// WARNING CODE //
	FB_AlarmCodeManager(
		bAlarm1			:= FALSE,   							//
		bAlarm2			:= FALSE, 								// 
		bAlarm3			:= FALSE, 								// 
		bAlarm4			:= FALSE, 								// 
		bAlarm5			:= FALSE,    							// 
		bAlarm6			:= FALSE, 								// 
		bAlarm7			:= FALSE, 								// 
		bAlarm8			:= FALSE, 								// 
		bAlarm9			:= FALSE,    							// 
		bAlarm10		:= FALSE, 								// 
		bAlarm11		:= FALSE, 								// 
		bAlarm12		:= FALSE, 								// 
		bAlarm13		:= FALSE,     							//
		bAlarm14		:= FALSE,  								//
		bAlarm15		:= FALSE,  								//
		wAlarmCode		=>MesDataExd.MesData.MesWarningCode);

// EVENT CODE //
	FB_AlarmCodeManager(
		bAlarm1			:= TON_Fermeture.Q AND NOT PT_Unlock_Alarm.Q, 	// Intrusion Detected
		bAlarm2			:= FALSE, 										// 
		bAlarm3			:= FALSE, 										// 
		bAlarm4			:= FALSE, 										// 
		bAlarm5			:= FALSE,    									// 
		bAlarm6			:= FALSE, 										// 
		bAlarm7			:= FALSE, 										// 
		bAlarm8			:= FALSE, 										// 
		bAlarm9			:= FALSE,    									// 
		bAlarm10		:= FALSE, 										// 
		bAlarm11		:= FALSE, 										// 
		bAlarm12		:= FALSE, 										// 
		bAlarm13		:= FALSE,     									// 
		bAlarm14		:= FALSE,  										// 
		bAlarm15		:= FALSE,  										// 
		wAlarmCode		=>MesDataExd.MesData.MesEventCode);
		
// When the alarm is activated for the first time, it is disabled for the duration of ParamTempoUnlockAlarm to avoid spamming alarms

PT_Unlock_Alarm(IN := TON_Fermeture.Q, PT := ParamTempoUnlockAlarm);
END_METHOD

METHOD M_Execute
//////////////////
//  Method Calls 
/////////////////

VAR 
	// Method local variables (reinitialized at each cycle) 
	
END_VAR

SUPER^.M_Execute() ;
END_METHOD

METHOD M_StateManager
//////////////////
// Detect when fire occurs
/////////////////

VAR 
	// Method local variables (reinitialized at each cycle)
 	MesStateInterm1 : BOOL;
	MesStateInterm2 : BOOL;
END_VAR

IF ParamCableCutSecurity THEN
	MesStateInterm1 := NOT IN_MesState1_IO ; 
	MesStateInterm2 := NOT IN_MesState2_IO ; 
ELSE 
	MesStateInterm1 := IN_MesState1_IO;
	MesStateInterm2 := IN_MesState2_IO;
END_IF

IF ParamNbSensors = 1 THEN 
	MesStateInterm2 := MesStateInterm1 ;
END_IF

IF ParamAtleastOne THEN 
MesDataExd.MesData.MesAlarmState := MesStateInterm1 OR MesStateInterm2 ; 
ELSE
MesDataExd.MesData.MesAlarmState := MesStateInterm1 AND MesStateInterm2 ; 
END_IF

R_TRIGAlarm(CLK:= MesDataExd.MesData.MesAlarmState ) ; 
IF R_TRIGAlarm.Q THEN
	MesCountAlarm :=  MIN(MesCountAlarm + 1 ,4294967295 ) ; 
ELSIF IN_ResetCounter THEN 
	MesCountAlarm := 0 ; 
END_IF

MesDataExd.MesData.MesCountAlarm	:= MesCountAlarm ;
END_METHOD

END_FUNCTION_BLOCK

// ---- 01_Equipement_Library/Sensors/TOR/FB_TOR_Spd.TcPOU
FUNCTION_BLOCK FB_TOR_Spd EXTENDS FB_TOR_Base
//////////////////
//  Surge Protection Device
//////////////////
VAR_INPUT PERSISTENT
	// Parameters of the Object (instance/model specific) 
	ParamTempoEs :TIME:=T#5S;(*  (s)Tempo before raising an alarm*)
END_VAR

VAR_OUTPUT
	//Child objects
	
END_VAR

VAR_INPUT
	// I/O Inputs 		                                     				
		
	
END_VAR

VAR
	//M_ALARMMANAGEMENT VARIABLES//
		FB_PermAlarm				: SR ;					// (NA) FB to maintain Fire Alarm even if sensor stop detection (burn) .
		TON_ES						: TON ; 
 
	//M_STATEMANAGER VARIABLES//
		MesDataExd			: TOR_Standard ;  

		
END_VAR

METHOD M_AlarmManagement
//////////////////
// Manages Smoke detector alarms and warnings
/////////////////

VAR 
	// Method local variables (reinitialized at each cycle) 
	FB_AlarmCodeManager			: FB_AlarmCodeManager ; 

END_VAR
// Detection Variables
TON_ES(IN:= MesDataExd.MesData.MesAlarmState , PT:= ParamTempoEs ) ; 
FB_PermAlarm(SET1 := TON_ES.Q  , Reset := CmdClearFault_G OR IN_CmdReset_L ); // SR FB for keep fire if burn .

// ALARM CODE //
	FB_AlarmCodeManager(
		bAlarm1			:= FB_PermAlarm.Q1 ,  														// Surge protection triggered	
		bAlarm2			:= SEL(ParamNbSensors=9,FALSE, IN_MesState1_IO <> IN_MesState2_IO), 		// UNcoherent measure
		bAlarm3			:=FALSE, 																	// 
		bAlarm4			:=FALSE, 																	// 
		bAlarm5			:=FALSE, 																	//	
		bAlarm6			:=FALSE,                                                                    //
		bAlarm7			:=FALSE,                                                                    //
		bAlarm8			:=FALSE,                                                                    //
		bAlarm9			:=FALSE,                                                                    //
		bAlarm10		:=FALSE,                                                                    //
		bAlarm11		:=FALSE,                                                                    //
		bAlarm12		:=FALSE,                                                                    //
		bAlarm13		:=FALSE,                                                                    //
		bAlarm14		:=FALSE,                                                                    //
		bAlarm15		:=FALSE,                                                                    //
		wAlarmCode		=>MesDataExd.MesData.MesAlarmCode );
		
// WARNING CODE //
	FB_AlarmCodeManager(
		bAlarm1			:= IN_MesState1_IO OR  IN_MesState2_IO,	  									// At least one detector is ON 
		bAlarm2			:=FALSE, 																	// 
		bAlarm3			:=FALSE, 																	// 
		bAlarm4			:=FALSE, 																	// 
		bAlarm5			:=FALSE, 																	//
		bAlarm6			:=FALSE,        															//
		bAlarm7			:=FALSE,        															//
		bAlarm8			:=FALSE,        															//
		bAlarm9			:=FALSE,        															//
		bAlarm10		:=FALSE,        															//
		bAlarm11		:=FALSE,        															//
		bAlarm12		:=FALSE,        															//
		bAlarm13		:=FALSE,        															//
		bAlarm14		:=FALSE,        															//
		bAlarm15		:=FALSE,        															//
		wAlarmCode			=>MesDataExd.MesData.MesWarningCode);
		
// EVENT CODE //
	FB_AlarmCodeManager(
		bAlarm1			:= IN_MesState1_IO, 															// First sensor is ON
		bAlarm2			:= IN_MesState2_IO, 															// Second sensor is ON
		bAlarm3			:= FALSE, 																		// 
		bAlarm4			:= FALSE, 																		// 
		bAlarm5			:= FALSE, 																		//			
		bAlarm6			:= FALSE,                           											//
		bAlarm7			:= FALSE,                           											//
		bAlarm8			:= FALSE,                           											//
		bAlarm9			:= FALSE,                           											//
		bAlarm10		:= FALSE,                           											//
		bAlarm11		:= FALSE,                           											//
		bAlarm12		:= FALSE,                           											//
		bAlarm13		:= FALSE,                           											//
		bAlarm14		:= FALSE,                           											//
		bAlarm15		:= FALSE,                           											//
		wAlarmCode		=>MesDataExd.MesData.MesEventCode);
END_METHOD

METHOD M_Execute
//////////////////
//  Method Calls 
/////////////////

VAR 
	// Method local variables (reinitialized at each cycle) 

END_VAR

	
	IF ParamNbSensors = 9 THEN // Use of contactor bi-stable No and NC
		IN_MesState2_IO := NOT IN_MesState2_IO;
	END_IF
SUPER^.M_Execute() ;
END_METHOD

METHOD M_StateManager
//////////////////
// Detect when fire occurs
/////////////////

VAR 
	// Method local variables (reinitialized at each cycle)
 	MesStateInterm1 : BOOL;
	MesStateInterm2 : BOOL;
END_VAR

IF ParamCableCutSecurity THEN
	MesStateInterm1 := NOT IN_MesState1_IO ; 
	MesStateInterm2 := NOT IN_MesState2_IO ; 
ELSE 
	MesStateInterm1 := IN_MesState1_IO;
	MesStateInterm2 := IN_MesState2_IO;
END_IF

IF ParamNbSensors = 1 THEN 
	MesStateInterm2 := MesStateInterm1 ;
END_IF

IF ParamAtleastOne THEN 
MesDataExd.MesData.MesAlarmState := MesStateInterm1 OR MesStateInterm2 ; 
ELSE
MesDataExd.MesData.MesAlarmState := MesStateInterm1 AND MesStateInterm2 ; 
END_IF

R_TRIGAlarm(CLK:= MesDataExd.MesData.MesAlarmState ) ; 
IF R_TRIGAlarm.Q THEN
	MesCountAlarm :=  MIN(MesCountAlarm + 1 ,4294967295 ) ; 
ELSIF IN_ResetCounter THEN 
	MesCountAlarm := 0 ; 
END_IF

MesDataExd.MesData.MesCountAlarm	:= MesCountAlarm ;
END_METHOD

END_FUNCTION_BLOCK

// ---- 01_Equipement_Library/Sensors/TOR/FB_TOR_VP.TcPOU
FUNCTION_BLOCK FB_TOR_VP EXTENDS FB_TOR_Base
//////////////////
//  Voltage Presence
//////////////////

VAR_INPUT PERSISTENT
	// Parameters of the Object (instance/model specific) 
		
		
END_VAR

VAR_OUTPUT
	//Child objects
	
END_VAR

VAR_INPUT
	// I/O Inputs 		                                     				
		
END_VAR

VAR
	//M_ALARMMANAGEMENT VARIABLES//
		
MesDataExd			: TOR_Standard ;  

	
END_VAR

METHOD M_AlarmManagement
//////////////////
// Manages Door sensor alarms and warnings
/////////////////

VAR 
	// Method local variables (reinitialized at each cycle) 
	FB_AlarmCodeManager : FB_AlarmCodeManager ; 


END_VAR

// ALARM CODE //
	FB_AlarmCodeManager(
 		bAlarm1			:= FALSE,    					// 
		bAlarm2			:= FALSE, 						// 
		bAlarm3			:= FALSE, 						// 
		bAlarm4			:= FALSE, 						// 
		bAlarm5			:= FALSE,       				//
		bAlarm6			:= FALSE,       				//
		bAlarm7			:= FALSE,       				//
		bAlarm8			:= FALSE,       				//
		bAlarm9			:= FALSE,       				//
		bAlarm10		:= FALSE,       				//
		bAlarm11		:= FALSE,       				//
		bAlarm12		:= FALSE,         				//
		bAlarm13		:= FALSE,         				//
		bAlarm14		:= FALSE,         				//
		bAlarm15		:= FALSE,         				//
		wAlarmCode		=>MesDataExd.MesData.MesAlarmCode);

// WARNING CODE //
	FB_AlarmCodeManager(
		bAlarm1			:= FALSE,    			// 
		bAlarm2			:= FALSE, 				//  
		bAlarm3			:= FALSE, 				//  
		bAlarm4			:= FALSE, 				//  
		bAlarm5			:= FALSE,               //
		bAlarm6			:= FALSE,               //
		bAlarm7			:= FALSE,               //
		bAlarm8			:= FALSE,               //
		bAlarm9			:= FALSE,               //
		bAlarm10		:= FALSE,               //
		bAlarm11		:= FALSE,               //
		bAlarm12		:= FALSE,               //
		bAlarm13		:= FALSE,               //
		bAlarm14		:= FALSE,               //
		bAlarm15		:= FALSE,               //
		wAlarmCode		=>MesDataExd.MesData.MesWarningCode);

// EVENT CODE //
	FB_AlarmCodeManager(
		bAlarm1			:= MesDataExd.MesData.MesAlarmState, 			//  Voltage not present anymore
		bAlarm2			:= FALSE, 							// 
		bAlarm3			:= FALSE, 							//  
		bAlarm4			:= FALSE, 							// 
		bAlarm5			:= FALSE,                           //
		bAlarm6			:= FALSE,                           //
		bAlarm7			:= FALSE,                           //
		bAlarm8			:= FALSE,                           //
		bAlarm9			:= FALSE,                           //
		bAlarm10		:= FALSE,                           //
		bAlarm11		:= FALSE,                           //
		bAlarm12		:= FALSE,                           //
		bAlarm13		:= FALSE,                           //
		bAlarm14		:= FALSE,                           //
		bAlarm15		:= FALSE,                           //
		wAlarmCode		=>MesDataExd.MesData.MesEventCode);
END_METHOD

METHOD M_StateManager
//////////////////
// Detect when fire occurs
/////////////////

VAR 
	// Method local variables (reinitialized at each cycle)
 	MesStateInterm1 : BOOL;
	MesStateInterm2 : BOOL;
END_VAR

IF ParamCableCutSecurity THEN
	MesStateInterm1 := NOT IN_MesState1_IO ; 
	MesStateInterm2 := NOT IN_MesState2_IO ; 
ELSE 
	MesStateInterm1 := IN_MesState1_IO;
	MesStateInterm2 := IN_MesState2_IO;
END_IF

IF ParamNbSensors = 1 THEN 
	MesStateInterm2 := MesStateInterm1 ;
END_IF

IF ParamAtleastOne THEN 
MesDataExd.MesData.MesAlarmState := MesStateInterm1 OR MesStateInterm2 ; 
ELSE
MesDataExd.MesData.MesAlarmState := MesStateInterm1 AND MesStateInterm2 ; 
END_IF

R_TRIGAlarm(CLK:= MesDataExd.MesData.MesAlarmState ) ; 
IF R_TRIGAlarm.Q THEN
	MesCountAlarm :=  MIN(MesCountAlarm + 1 ,4294967295 ) ; 
ELSIF IN_ResetCounter THEN 
	MesCountAlarm := 0 ; 
END_IF

MesDataExd.MesData.MesCountAlarm	:= MesCountAlarm ;
END_METHOD

END_FUNCTION_BLOCK

// ---- 01_Equipement_Library/Sensors/TOR/FB_TOR_DS.TcPOU
FUNCTION_BLOCK FB_TOR_DS EXTENDS FB_TOR_Base
//////////////////
//  Door sensor system . State = True >> Door Closed .
//////////////////

VAR_INPUT PERSISTENT
	// Parameters of the Object (instance/model specific) 
		ParamTempoDoorAlarm			: TIME := T#10S ;	(* (s) Tempo for Door sensor alarm *)
		
END_VAR

VAR_OUTPUT
	//Child objects
	
END_VAR

VAR_INPUT
	// I/O Inputs 		                                     				
		
END_VAR

VAR
	//M_ALARMMANAGEMENT VARIABLES//
		TON_Ouverture				: TON;				//(NA) Tempo to detect door opened for too long time . 
	MesDataExd			: TOR_Standard ;  



END_VAR

METHOD M_AlarmManagement
//////////////////
// Manages Door sensor alarms and warnings
/////////////////

VAR 
	// Method local variables (reinitialized at each cycle) 
	FB_AlarmCodeManager : FB_AlarmCodeManager ; 


END_VAR
// Detection Variables
TON_Ouverture(IN:= MesDataExd.MesData.MesAlarmState,PT:=ParamTempoDoorAlarm);

// ALARM CODE //
	FB_AlarmCodeManager(
 		bAlarm1			:= FALSE,    	// 
		bAlarm2			:= FALSE, 		// 
		bAlarm3			:= FALSE, 		// 
		bAlarm4			:= FALSE, 		// 
		bAlarm5			:= FALSE,       //
		bAlarm6			:= FALSE,       //
		bAlarm7			:= FALSE,       //
		bAlarm8			:= FALSE,       //
		bAlarm9			:= FALSE,       //
		bAlarm10		:= FALSE,       //
		bAlarm11		:= FALSE,       //
		bAlarm12		:= FALSE,       //
		bAlarm13		:= FALSE,       //
		bAlarm14		:= FALSE,       //
		bAlarm15		:= FALSE,       //
		wAlarmCode		=>MesDataExd.MesData.MesAlarmCode);

// WARNING CODE //
	FB_AlarmCodeManager(
		bAlarm1			:= TON_Ouverture.Q,    	// The door is open for more than 15 seconds
		bAlarm2			:= FALSE, 				// 
		bAlarm3			:= FALSE, 				// 
		bAlarm4			:= FALSE, 				// 
		bAlarm5			:= FALSE, 				//
		bAlarm6			:= FALSE,               //
		bAlarm7			:= FALSE,               //
		bAlarm8			:= FALSE,               //
		bAlarm9			:= FALSE,               //
		bAlarm10		:= FALSE,               //
		bAlarm11		:= FALSE,               //
		bAlarm12		:= FALSE,               //
		bAlarm13		:= FALSE,               //
		bAlarm14		:= FALSE,               //
		bAlarm15		:= FALSE,               //
		wAlarmCode		=>MesDataExd.MesData.MesWarningCode);

// EVENT CODE //
	FB_AlarmCodeManager(
		bAlarm1			:= MesDataExd.MesData.MesAlarmState, 		// Door is Opened
		bAlarm2			:= FALSE, 						// 
		bAlarm3			:= FALSE, 						// 
		bAlarm4			:= FALSE, 						// 
		bAlarm5			:= FALSE, 						//
		bAlarm6			:= FALSE, 						//
		bAlarm7			:= FALSE, 						//
		bAlarm8			:= FALSE, 						//
		bAlarm9			:= FALSE, 						//
		bAlarm10		:= FALSE, 						//
		bAlarm11		:= FALSE, 						//
		bAlarm12		:= FALSE, 						//
		bAlarm13		:= FALSE, 						//
		bAlarm14		:= FALSE, 						//
		bAlarm15		:= FALSE, 						//
		wAlarmCode		=>MesDataExd.MesData.MesEventCode);
END_METHOD

METHOD M_Execute
//////////////////
//  Method Calls 
/////////////////

VAR 
	// Method local variables (reinitialized at each cycle) 
	
END_VAR


SUPER^.M_Execute() ;
END_METHOD

METHOD M_StateManager
//////////////////
// Detect when fire occurs
/////////////////

VAR 
	// Method local variables (reinitialized at each cycle)
 	MesStateInterm1 : BOOL;
	MesStateInterm2 : BOOL;
END_VAR

IF ParamCableCutSecurity THEN
	MesStateInterm1 := NOT IN_MesState1_IO ; 
	MesStateInterm2 := NOT IN_MesState2_IO ; 
ELSE 
	MesStateInterm1 := IN_MesState1_IO;
	MesStateInterm2 := IN_MesState2_IO;
END_IF

IF ParamNbSensors = 1 THEN 
	MesStateInterm2 := MesStateInterm1 ;
END_IF

IF ParamAtleastOne THEN 
MesDataExd.MesData.MesAlarmState := MesStateInterm1 OR MesStateInterm2 ; 
ELSE
MesDataExd.MesData.MesAlarmState := MesStateInterm1 AND MesStateInterm2 ; 
END_IF

R_TRIGAlarm(CLK:= MesDataExd.MesData.MesAlarmState ) ; 
IF R_TRIGAlarm.Q THEN
	MesCountAlarm :=  MIN(MesCountAlarm + 1 ,4294967295 ) ; 
ELSIF IN_ResetCounter THEN 
	MesCountAlarm := 0 ; 
END_IF

MesDataExd.MesData.MesCountAlarm	:= MesCountAlarm ;
END_METHOD

END_FUNCTION_BLOCK

// ---- 01_Equipement_Library/Sensors/TOR/FB_TOR_Rain.TcPOU
FUNCTION_BLOCK FB_TOR_Rain EXTENDS FB_TOR_Base
//////////////////
//  Rain sensor system.
//////////////////

VAR_INPUT PERSISTENT
	// Parameters of the Object (instance/model specific) 
	ParamRainPerPulse				: REAL := 10 ; (* (mm) Number of mm of rain per pulse		*)
END_VAR

VAR_OUTPUT
	//Child objects
	
END_VAR

VAR_INPUT
	// I/O Inputs 		                                     				
    ParamVarHrWarning   			: REAL :=8 ;  // (mm) Max of raining before warning mm of rain for last hour --> Mean it is raining a lot  Defaut value 8       
    ParamVarDayWarning  			: REAL :=48;  // (mm )max of raining before warning mm of rain for last day  --> Mean it rained a lot during 1 day defaut value 48
	ParamVarMinAlarm				: REAL :=-5;  // (%)  Config : Minimal allowed Site Hygrometry 
END_VAR

VAR
	MesDataExd			: TOR_Rain;

	//M_ALARMMANAGEMENT VARIABLES//
		WarningDay					: BOOL;
		WarningHr					: BOOL;
		WarningValue				: BOOL;
	
	
	//M_Execute
		FB_AverageHr				: FB_Average; 	
	    FB_AverageDay               : FB_Average;
	    FB_AverageMonth             : FB_Average;
		CTUHr						: CTU;
		CTUDay						: CTU;
		CTUMonth					: CTU;
		Hour 						: INT;
		PluvioHr_Avg		        : REAL ; 
		PluvioDay_Avg		        : REAL ; 
		PluvioMonth_Avg		        : REAL ;     
		PluvioHr_Max		        : REAL;
		PluvioDay_Max		        : REAL ; 
		PluvioMonth_Max		        : REAL ; 
        PluvioHr					: REAL ; 
		PluvioDay					: REAL ; 
		PluvioMonth					: REAL ; 

	
	
END_VAR

METHOD M_AlarmManagement
//////////////////
// Manages Door sensor alarms and warnings
/////////////////

VAR 
	// Method local variables (reinitialized at each cycle) 
	FB_AlarmCodeManager : FB_AlarmCodeManager ; 
END_VAR
	WarningDay	:= PluvioDay >= ParamVarDayWarning;
	WarningHr	:= PluvioHr >= ParamVarHrWarning;
	WarningValue:= PluvioDay <= ParamVarMinAlarm OR PluvioHr <= ParamVarMinAlarm;

// ALARM CODE //
	FB_AlarmCodeManager(
 		bAlarm1			:= FALSE,    								// 
		bAlarm2			:= FALSE, 									// 
		bAlarm3			:= FALSE, 									// 
		bAlarm4			:= FALSE, 									// 
		bAlarm5			:= FALSE,     								//
		bAlarm6			:= FALSE,  									//
		bAlarm7			:= FALSE,  									//
		bAlarm8			:= FALSE,  									//
		bAlarm9			:= FALSE,    								// 
		bAlarm10		:= FALSE, 									// 
		bAlarm11		:= FALSE, 									// 
		bAlarm12		:= FALSE, 									// 
		bAlarm13		:= FALSE,									// 
		bAlarm14		:= FALSE,									// 
		bAlarm15		:= FALSE,									// 
		wAlarmCode		=>MesDataExd.MesData.MesAlarmCode);

// WARNING CODE //
	FB_AlarmCodeManager(
		bAlarm1			:= WarningHr,   							// Raining too hard 
		bAlarm2			:= WarningDay, 								// Raining a lot during one day
		bAlarm3			:= WarningValue, 							// Raining value not coherent
		bAlarm4			:= FALSE, 									// 
		bAlarm5			:= FALSE,    								// 
		bAlarm6			:= FALSE, 									// 
		bAlarm7			:= FALSE, 									// 
		bAlarm8			:= FALSE, 									// 
		bAlarm9			:= FALSE,    								// 
		bAlarm10		:= FALSE, 									// 
		bAlarm11		:= FALSE, 									// 
		bAlarm12		:= FALSE, 									// 
		bAlarm13		:= FALSE,									// 
		bAlarm14		:= FALSE,									// 
		bAlarm15		:= FALSE,									// 
		wAlarmCode		=>MesDataExd.MesData.MesWarningCode);

// EVENT CODE //
	FB_AlarmCodeManager(
		bAlarm1			:= MesDataExd.MesData.MesAlarmState, 		// 0.2mm of water falled
		bAlarm2			:= FALSE, 									// 
		bAlarm3			:= FALSE, 									// 
		bAlarm4			:= FALSE, 									// 
		bAlarm5			:= FALSE, 									// 
		bAlarm6			:= FALSE, 									// 
		bAlarm7			:= FALSE, 									// 
		bAlarm8			:= FALSE, 									// 
		bAlarm9			:= FALSE, 									// 
		bAlarm10		:= FALSE, 									// 
		bAlarm11		:= FALSE, 									// 
		bAlarm12		:= FALSE, 									// 
		bAlarm13		:= FALSE, 									// 
		bAlarm14		:= FALSE, 									//  
		bAlarm15		:= FALSE, 									//  
		wAlarmCode		=>MesDataExd.MesData.MesEventCode);
END_METHOD

METHOD M_Execute
//////////////////
//  Method Calls 
/////////////////

VAR 
	// Method local variables (reinitialized at each cycle) 
	
END_VAR
// EMULATOR I/O //

//MAIN CODE HERE
Hour 							:=CstCycleTime_G/1000/3600  ;                        

CTUHr   (CU:= MesDataExd.MesData.MesAlarmState , RESET :=  Hour MOD 1 = 0) ; 
CTUDay  (CU:= MesDataExd.MesData.MesAlarmState , RESET := Hour MOD 24 = 0 ) ; 
CTUMonth(CU:= MesDataExd.MesData.MesAlarmState , RESET := Hour MOD 24*30 = 0 ) ; 

PluvioHr_Max := SEL( Hour MOD 1 = 0  ,   PluvioHr_Max , PluvioHr_Max:= PluvioHr)  ; 
PluvioHr := CTUHr.CV * ParamRainPerPulse ; 

PluvioDay_Max := SEL( Hour MOD 24 = 0  ,   PluvioDay_Max , PluvioDay_Max:= PluvioDay)  ; 
PluvioDay := CTUDay.CV * ParamRainPerPulse ; 

PluvioMonth_Max := SEL( Hour MOD 24*30 = 0  ,   PluvioMonth_Max , PluvioMonth_Max:= PluvioMonth)  ; 
PluvioMonth := CTUMonth.CV * ParamRainPerPulse ; 


//FB_AverageHr(ValueIn:=PluvioHr_Max  , WindowDuration := 24*3600*1000 , ValueOut => PluvioHr_Avg) ; 
//FB_AverageDay(ValueIn:=PluvioDay_Max  , WindowDuration := 24*30*3600*1000 , ValueOut => PluvioDay_Avg) ; 
//FB_AverageMonth(ValueIn:=PluvioMonth_Max  , WindowDuration := 24*365*3600*1000 , ValueOut => PluvioMonth_Avg) ;
//EVALUATE

MesDataExd.MesRainFall_LastHour 	:= PluvioHr;
MesDataExd.MesRainFall_LastDay		:= PluvioDay;
MesDataExd.MesRainFall_LastMonth	:= PluvioMonth;
MesDataExd.AvgmmHour				:= PluvioHr_Avg;
MesDataExd.AvgmmDay					:= PluvioDay_Avg;
MesDataExd.AvgmmMonth				:= PluvioMonth_Avg;

SUPER^.M_Execute();
END_METHOD

METHOD M_StateManager
//////////////////
// Detect when fire occurs
/////////////////

VAR 
	// Method local variables (reinitialized at each cycle)
 	MesStateInterm1 : BOOL;
	MesStateInterm2 : BOOL;
END_VAR

IF ParamCableCutSecurity THEN
	MesStateInterm1 := NOT IN_MesState1_IO ; 
	MesStateInterm2 := NOT IN_MesState2_IO ; 
ELSE 
	MesStateInterm1 := IN_MesState1_IO;
	MesStateInterm2 := IN_MesState2_IO;
END_IF

IF ParamNbSensors = 1 THEN 
	MesStateInterm2 := MesStateInterm1 ;
END_IF

IF ParamAtleastOne THEN 
MesDataExd.MesData.MesAlarmState := MesStateInterm1 OR MesStateInterm2 ; 
ELSE
MesDataExd.MesData.MesAlarmState := MesStateInterm1 AND MesStateInterm2 ; 
END_IF

R_TRIGAlarm(CLK:= MesDataExd.MesData.MesAlarmState ) ; 
IF R_TRIGAlarm.Q THEN
	MesCountAlarm :=  MIN(MesCountAlarm + 1 ,4294967295 ) ; 
ELSIF IN_ResetCounter THEN 
	MesCountAlarm := 0 ; 
END_IF

MesDataExd.MesData.MesCountAlarm	:= MesCountAlarm ;
END_METHOD

END_FUNCTION_BLOCK

// ---- 01_Equipement_Library/Sensors/TOR/FB_TOR_SD.TcPOU
FUNCTION_BLOCK FB_TOR_SD EXTENDS FB_TOR_Base
//////////////////
//  Smoke and Fire detection system with Typhoon triggering system. 
//////////////////
VAR_INPUT PERSISTENT
	// Parameters of the Object (instance/model specific) 
	ParamTempoFire :TIME:=T#2S;(*  (s)Tempo before raising an alarm*)
END_VAR

VAR_OUTPUT
	//Child objects
	
END_VAR

VAR_INPUT
	// I/O Inputs 		                                     				
		
		MesDataExd			: TOR_Standard ;  

END_VAR

VAR
	//M_ALARMMANAGEMENT VARIABLES//
		FB_PermAlarm				: SR ;					// (NA) FB to maintain Fire Alarm even if sensor stop detection (burn) .
		TON_Fire					: TON ; 
 
	//M_STATEMANAGER VARIABLES//
		
END_VAR

METHOD M_AlarmManagement
//////////////////
// Manages Smoke detector alarms and warnings
/////////////////

VAR 
	// Method local variables (reinitialized at each cycle) 
	FB_AlarmCodeManager			: FB_AlarmCodeManager ; 

END_VAR
// Detection Variables
TON_Fire(IN:= MesDataExd.MesData.MesAlarmState , PT:= ParamTempoFire ) ; 
FB_PermAlarm(SET1 := TON_Fire.Q  , Reset := CmdClearFault_G OR IN_CmdReset_L ); // SR FB for keep fire if burn .

// ALARM CODE //
	FB_AlarmCodeManager(
		bAlarm1			:= FB_PermAlarm.Q1 ,  				// Fire detection		
		bAlarm2			:=FALSE, 							// 
		bAlarm3			:=FALSE, 							// 
		bAlarm4			:=FALSE, 							// 
		bAlarm5			:=FALSE, 							//
		bAlarm6			:=FALSE,                            //
		bAlarm7			:=FALSE,                            //
		bAlarm8			:=FALSE,                            //
		bAlarm9			:=FALSE,                            //
		bAlarm10		:=FALSE,                            //
		bAlarm11		:=FALSE,                            //
		bAlarm12		:=FALSE,                            //
		bAlarm13		:=FALSE,                            //
		bAlarm14		:=FALSE,                            //
		bAlarm15		:=FALSE,                            //
		wAlarmCode		=>MesDataExd.MesData.MesAlarmCode );
		
// WARNING CODE //
	FB_AlarmCodeManager(
		bAlarm1			:= FALSE,	  															//  
		bAlarm2			:= FALSE, 																//
		bAlarm3			:=FALSE, 																// 
		bAlarm4			:=FALSE, 																// 
		bAlarm5			:=FALSE, 																// 
		bAlarm6			:=FALSE,                                                                //
		bAlarm7			:=FALSE,                                                                //
		bAlarm8			:=FALSE,                                                                //
		bAlarm9			:=FALSE,                                                                //
		bAlarm10		:=FALSE,                                                                //
		bAlarm11		:=FALSE,                                                                //
		bAlarm12		:=FALSE,                                                                //
		bAlarm13		:=FALSE,                                                                //
		bAlarm14		:=FALSE,                                                                //
		bAlarm15		:=FALSE,                                                                //
		wAlarmCode		=>MesDataExd.MesData.MesWarningCode);
		
// EVENT CODE //
	FB_AlarmCodeManager(
		bAlarm1			:= FALSE,
		bAlarm2			:= FALSE,
		bAlarm3			:= FALSE, 					// 		
		bAlarm4			:= FALSE, 					// 
		bAlarm5			:= FALSE, 					//
		bAlarm6			:= FALSE,                   //
		bAlarm7			:= FALSE,                   //
		bAlarm8			:= FALSE,                   //
		bAlarm9			:= FALSE,                   //
		bAlarm10		:= FALSE,                   //
		bAlarm11		:= FALSE,                   //
		bAlarm12		:= FALSE,                   //
		bAlarm13		:= FALSE,                   //
		bAlarm14		:= FALSE,                   //
		bAlarm15		:= FALSE,                   //
		wAlarmCode		=>MesDataExd.MesData.MesEventCode);
END_METHOD

METHOD M_Execute
//////////////////
//  Method Calls 
/////////////////

VAR 
	// Method local variables (reinitialized at each cycle) 

END_VAR

	IF ParamNbSensors = 9 THEN // Use of contactor bi-stable No and NC
		IN_MesState2_IO := NOT IN_MesState2_IO;
	END_IF
SUPER^.M_Execute() ;
END_METHOD

METHOD M_StateManager
//////////////////
// Detect when fire occurs
/////////////////

VAR 
	// Method local variables (reinitialized at each cycle)
 	MesStateInterm1 : BOOL;
	MesStateInterm2 : BOOL;
END_VAR

IF ParamCableCutSecurity THEN
	MesStateInterm1 := NOT IN_MesState1_IO ; 
	MesStateInterm2 := NOT IN_MesState2_IO ; 
ELSE 
	MesStateInterm1 := IN_MesState1_IO;
	MesStateInterm2 := IN_MesState2_IO;
END_IF

IF ParamNbSensors = 1 THEN 
	MesStateInterm2 := MesStateInterm1 ;
END_IF

IF ParamAtleastOne THEN 
MesDataExd.MesData.MesAlarmState := MesStateInterm1 OR MesStateInterm2 ; 
ELSE
MesDataExd.MesData.MesAlarmState := MesStateInterm1 AND MesStateInterm2 ; 
END_IF

R_TRIGAlarm(CLK:= MesDataExd.MesData.MesAlarmState ) ; 
IF R_TRIGAlarm.Q THEN
	MesCountAlarm :=  MIN(MesCountAlarm + 1 ,4294967295 ) ; 
ELSIF IN_ResetCounter THEN 
	MesCountAlarm := 0 ; 
END_IF

MesDataExd.MesData.MesCountAlarm	:= MesCountAlarm ;
END_METHOD

END_FUNCTION_BLOCK

// ---- 01_Equipement_Library/Sensors/TOR/FB_TOR_ToS.TcPOU
FUNCTION_BLOCK FB_TOR_ToS EXTENDS FB_TOR_Base
//////////////////
//  Technician on site selectOR   
//////////////////

VAR_INPUT PERSISTENT
	// Parameters of the Object (instance/model specific) 
	ParamTempoToSAlarm				: TIME := T#180M ; 	(*(min) Tempo (2h30) after ToS without clear fault >> alarm *)
	ParamTempoToSWarning			: TIME := T#120M ;  (* (min) Tempo (2h) after ToS without clear fault  >> warning*)
END_VAR

VAR_OUTPUT
	//Child objects
	
END_VAR

VAR_INPUT
	// I/O Inputs 		                                     				
	
END_VAR

VAR
	//M_ALARMMANAGEMENT VARIABLES//
		TON 						: TON ;  			 // (NA) Calculate time since technician presence activation. 
		        
MesDataExd			: TOR_Standard ;                              			
	          	

	

		
END_VAR

METHOD M_AlarmManagement
//////////////////
// Manages Smoke detector alarms and warnings
/////////////////

VAR 
	// Method local variables (reinitialized at each cycle) 
	FB_AlarmCodeManager : FB_AlarmCodeManager ; 
	
END_VAR
// Detection Variables
	TON(IN:= MesDataExd.MesData.MesAlarmState AND NOT CmdClearFault_G , PT:=ParamTempoToSAlarm);   			// Reset tempo if reset commAND  
	
// ALARM CODE //
	FB_AlarmCodeManager(
		bAlarm1			:= TON.Q ,													// If technician presence is active for more than 6 hours . 				
		bAlarm2			:=FALSE, 													// 
		bAlarm3			:=FALSE, 													// 
		bAlarm4			:=FALSE, 													// 
		bAlarm5			:=FALSE, 													//
		bAlarm6			:=FALSE,        											//
		bAlarm7			:=FALSE,        											//
		bAlarm8			:=FALSE,        											//
		bAlarm9			:=FALSE,        											//
		bAlarm10		:=FALSE,        											//
		bAlarm11		:=FALSE,        											//
		bAlarm12		:=FALSE,        											//
		bAlarm13		:=FALSE,        											//
		bAlarm14		:=FALSE,        											//
		bAlarm15		:=FALSE,        											//
		wAlarmCode		=>MesDataExd.MesData.MesAlarmCode);

// WARNING CODE //
	FB_AlarmCodeManager(
		bAlarm1			:= TON.ET > ParamTempoToSWarning ,				// If technician presence is active for more than 2 hours .  
		bAlarm2			:=FALSE, 										// 
		bAlarm3			:=FALSE, 										// 
		bAlarm4			:=FALSE, 										// 
		bAlarm5			:=FALSE, 										//
		bAlarm6			:=FALSE,        								//
		bAlarm7			:=FALSE,        								//
		bAlarm8			:=FALSE,        								//
		bAlarm9			:=FALSE,        								//
		bAlarm10		:=FALSE,        								//
		bAlarm11		:=FALSE,        								//
		bAlarm12		:=FALSE,        								//
		bAlarm13		:=FALSE,        								//
		bAlarm14		:=FALSE,        								//
		bAlarm15		:=FALSE,        								//
		wAlarmCode		=>MesDataExd.MesData.MesWarningCode);
			
// EVENT CODE //
	FB_AlarmCodeManager(
		bAlarm1			:= MesDataExd.MesData.MesAlarmState, 		// Technician On Site
		bAlarm2			:= FALSE, 						// 
		bAlarm3			:= FALSE, 						// 
		bAlarm4			:= FALSE, 						// 
		bAlarm5			:= FALSE, 						//
		bAlarm6			:= FALSE, 						//
		bAlarm7			:= FALSE,                       //
		bAlarm8			:= FALSE,                       //
		bAlarm9			:= FALSE,                       //
		bAlarm10		:= FALSE,                       //
		bAlarm11		:= FALSE,                       //
		bAlarm12		:= FALSE,                       //
		bAlarm13		:= FALSE,                       //
		bAlarm14		:= FALSE,                       //
		bAlarm15		:= FALSE,                       //
		wAlarmCode		=>MesDataExd.MesData.MesEventCode);
END_METHOD

METHOD M_Execute
//////////////////
//  Method Calls 
/////////////////

VAR 
	// Method local variables (reinitialized at each cycle) 

END_VAR
// EMULATOR I/O //

SUPER^.M_Execute() ;
END_METHOD

METHOD M_StateManager
//////////////////
// Detect when fire occurs
/////////////////

VAR 
	// Method local variables (reinitialized at each cycle)
 	MesStateInterm1 : BOOL;
	MesStateInterm2 : BOOL;
END_VAR

IF ParamCableCutSecurity THEN
	MesStateInterm1 := NOT IN_MesState1_IO ; 
	MesStateInterm2 := NOT IN_MesState2_IO ; 
ELSE 
	MesStateInterm1 := IN_MesState1_IO;
	MesStateInterm2 := IN_MesState2_IO;
END_IF

IF ParamNbSensors = 1 THEN 
	MesStateInterm2 := MesStateInterm1 ;
END_IF

IF ParamAtleastOne THEN 
MesDataExd.MesData.MesAlarmState := MesStateInterm1 OR MesStateInterm2 ; 
ELSE
MesDataExd.MesData.MesAlarmState := MesStateInterm1 AND MesStateInterm2 ; 
END_IF

R_TRIGAlarm(CLK:= MesDataExd.MesData.MesAlarmState ) ; 
IF R_TRIGAlarm.Q THEN
	MesCountAlarm :=  MIN(MesCountAlarm + 1 ,4294967295 ) ; 
ELSIF IN_ResetCounter THEN 
	MesCountAlarm := 0 ; 
END_IF

MesDataExd.MesData.MesCountAlarm	:= MesCountAlarm ;
END_METHOD

END_FUNCTION_BLOCK

// ---- 01_Equipement_Library/Tariff Meter/FB_EM_Base.TcPOU
FUNCTION_BLOCK FB_EM_Base
//////////////////
// Measurement Solution. Base FB
//////////////////
VAR_INPUT PERSISTENT
	// Parameters of the Object (instance specific) 
		CmdInitialValues			: EM_Standard;
	{attribute 'OPC.UA.DA' := '1'} 
		ParamStepEactCons			: REAL := 10;	// kWh step for tariff meter
	{attribute 'OPC.UA.DA' := '1'}                  
		ParamStepEactProd			: REAL := 10;   // kWh step for tariff meter
	{attribute 'OPC.UA.DA' := '1'}                  
		ParamStepEreactCons			: REAL := 10;   // kVArh step for tariff meter
	{attribute 'OPC.UA.DA' := '1'}                  
		ParamStepEreactProd			: REAL := 10;   // kVArh step for tariff meter
		ParamEssNum					: UINT :=1 ; 	// ESS Num
END_VAR

VAR_INPUT
	//Child objects
		IN_CmdReset_L					: BOOL;			// (NA) Local reset of the alarms	
END_VAR                                                             
VAR                                                                 
	//M_ALARMMANAGEMENT VARIABLES//                                 
		TON_ComAlarm				: TON ; 			// Tempo before deteting loss of communication. 
                                                        
	//M_INIT VARIABLES //                               
		bInit						: BOOL 	:= TRUE ; 	// (NA) Initialize object parameters at first cycle 
		                                                
	// M_EXECUTE VARIABLES //                           
 //	MesDataExd			: EM;					// (NA) Structure of the Tariff Meter
		MesCP_Read					: BOOL := TRUE;	(* Read function enable *)
		MesCP_Write					: BOOL := TRUE;	(* Write function enable *)                                                
	// M_EVALUATE VARIABLES //                          
		trig1 						: R_TRIG;			// (NA) Trigger for the pulses
		trig2 						: R_TRIG;			// (NA) Trigger for the pulses
		trig3 						: R_TRIG;			// (NA) Trigger for the pulses
		trig4 						: R_TRIG;			// (NA) Trigger for the pulses

                      
END_VAR

VAR_INPUT
		IN_MesPulseEactCons_IO			: BOOL;		// Pulse Input signal for the Active energy consumed measurement
		IN_MesPulseEactProd_IO			: BOOL;		// Pulse Input signal for the Active energy produced measurement
		IN_MesPulseEreactCons_IO		: BOOL;		// Pulse Input signal for the Reactive energy consumed measurement
		IN_MesPulseEreactProd_IO		: BOOL;		// Pulse Input signal for the Reactive energy produced measurement
END_VAR

METHOD M_AlarmManagement
//////////////////
// Digiware measurement tool alarm and warning management
/////////////////

VAR 
	
END_VAR
END_METHOD

METHOD M_Evaluate
VAR_INPUT
END_VAR

VAR

END_VAR
END_METHOD

METHOD M_Execute
//////////////////
//  Method Calls 
/////////////////
VAR 
	// Method local variables (reinitialized at each cycle) 
	// EMULATOR

	
END_VAR



// METHODS CALLS //
	IF bInit THEN
		M_Init() ; 
		bInit					:= FALSE ; 
	ELSIF CmdClearFault_G OR IN_CmdReset_L THEN 
		bInit:= TRUE ;
	END_IF

	M_Evaluate();	

	////////////////////
	M_AlarmManagement();
END_METHOD

METHOD M_Init
VAR 

END_VAR
END_METHOD

END_FUNCTION_BLOCK

// ---- 01_Equipement_Library/Tariff Meter/FB_EM_Pulse.TcPOU
FUNCTION_BLOCK FB_EM_Pulse EXTENDS FB_EM_Base
//////////////////
// Measurement Solution. Base FB
//////////////////
VAR_INPUT PERSISTENT
	// Parameters of the Object (instance specific) 
		
	
END_VAR

VAR_OUTPUT
	//Child objects
	
END_VAR
VAR
	//M_ALARMMANAGEMENT VARIABLES//
		FB_DetectFixedValue   : FB_DetectFixedValue ; 
        Eact_null    		  : REAL ;                                   								
		

	//M_INIT VARIABLES //
		MesDataExd			: EM_Standard ; 
		
	// M_EXECUTE VARIABLES //
 		
	// M_Reset_L
		
                      
END_VAR

VAR_INPUT
		
END_VAR

METHOD M_AlarmManagement
//////////////////
// Digiware measurement tool alarm and warning management
/////////////////

VAR 
	FB_AlarmCodeManager : FB_AlarmCodeManager ; 
END_VAR

FB_DetectFixedValue(IN_Addr := ADR(MesDataExd.MesData.MesEactCons) , IN_Size := SIZEOF(MesDataExd.MesData.MesEactCons) , IN_Duration :=T#3H , IN_EmptyStruct := ADR(Eact_null ) ); 

// ALARM CODE //
	FB_AlarmCodeManager(
		bAlarm1			:= MesDataExd.MesData.MesEActProd > 10 ,																			// Production measured			
		bAlarm2			:=FB_DetectFixedValue.OUT_bStatic 	,																	// Loss of communication with meter 
		bAlarm3			:=FALSE, 																								// 
		bAlarm4			:=FALSE, 																								// 
		bAlarm5			:=FALSE, 																								//
		bAlarm6			:=FALSE,        																						//
		bAlarm7			:=FALSE,        																						//
		bAlarm8			:=FALSE,        																						//
		bAlarm9			:=FALSE,        																						//
		bAlarm10		:=FALSE,        																						//
		bAlarm11		:=FALSE,        																						//
		bAlarm12		:=FALSE,        																						//
		bAlarm13		:=FALSE,        																						//
		bAlarm14		:=FALSE,        																						//
		bAlarm15		:=FALSE,        																						//
		wAlarmCode		=>MesDataExd.MesData.MesAlarmCode);

// WARNING CODE //

	FB_AlarmCodeManager(
		bAlarm1			:= FALSE ,										//  
		bAlarm2			:=FALSE, 										// 
		bAlarm3			:=FALSE, 										// 
		bAlarm4			:=FALSE, 										// 
		bAlarm5			:=FALSE, 										//
		bAlarm6			:=FALSE,        								//
		bAlarm7			:=FALSE,        								//
		bAlarm8			:=FALSE,        								//
		bAlarm9			:=FALSE,        								//
		bAlarm10		:=FALSE,        								//
		bAlarm11		:=FALSE,        								//
		bAlarm12		:=FALSE,        								//
		bAlarm13		:=FALSE,        								//
		bAlarm14		:=FALSE,        								//
		bAlarm15		:=FALSE,        								//
		wAlarmCode		=>MesDataExd.MesData.MesWarningCode);
			
// EVENT CODE //
	FB_AlarmCodeManager(
		bAlarm1			:= IN_CmdReset_L, 				// Reset command
		bAlarm2			:= FALSE, 						// 
		bAlarm3			:= FALSE, 						// 
		bAlarm4			:= FALSE, 						// 
		bAlarm5			:= FALSE, 						//
		bAlarm6			:= FALSE, 						//
		bAlarm7			:= FALSE,                       //
		bAlarm8			:= FALSE,                       //
		bAlarm9			:= FALSE,                       //
		bAlarm10		:= FALSE,                       //
		bAlarm11		:= FALSE,                       //
		bAlarm12		:= FALSE,                       //
		bAlarm13		:= FALSE,                       //
		bAlarm14		:= FALSE,                       //
		bAlarm15		:= FALSE,                       //
		wAlarmCode		=>MesDataExd.MesData.MesEventCode);
END_METHOD

METHOD M_Evaluate
VAR_INPUT
END_VAR

VAR
	TM_0 : EM_Standard;	// Empty structure
	OutTrig_Eac : BOOL;
	OutTrig_Eap : BOOL;
	OutTrig_Erc : BOOL;
	OutTrig_Erp : BOOL;
	bTest : BOOL;
END_VAR
IF CmdInitialValues.MesData.MesEactCons <> TM_0.MesData.MesEactCons OR CmdInitialValues.MesData.MesEActProd <> TM_0.MesData.MesEActProd OR CmdInitialValues.MesData.MesEReactCons <> TM_0.MesData.MesEReactCons OR CmdInitialValues.MesData.MesEReactProd <> TM_0.MesData.MesEReactProd THEN
MesDataExd:= CmdInitialValues;
	CmdInitialValues := TM_0 ;
END_IF

trig1(CLK := IN_MesPulseEactCons_IO, Q => OutTrig_Eac);
trig2(CLK := IN_MesPulseEactProd_IO, Q => OutTrig_Eap);
trig3(CLK:= IN_MesPulseEreactCons_IO, Q => OutTrig_Erc);
trig4(CLK:= IN_MesPulseEreactProd_IO, Q => OutTrig_Erp);

IF OutTrig_Eac THEN
MesDataExd.MesData.MesEactCons := MesDataExd.MesData.MesEactCons + ParamStepEactCons;
END_IF 

IF OutTrig_Eap THEN
MesDataExd.MesData.MesEActProd := MesDataExd.MesData.MesEActProd + ParamStepEactProd;
END_IF 

IF OutTrig_Erc THEN
MesDataExd.MesData.MesEReactCons := MesDataExd.MesData.MesEReactCons + ParamStepEreactCons;
END_IF 

IF OutTrig_Erp THEN
MesDataExd.MesData.MesEReactProd := MesDataExd.MesData.MesEReactProd + ParamStepEreactProd;
END_IF 

SUPER^.M_Evaluate();
END_METHOD

METHOD M_Init
VAR 
	InitialValues : EM_Standard ; 
END_VAR
MesDataExd := InitialValues ; 
bInit := FALSE ;
END_METHOD

END_FUNCTION_BLOCK

// ---- 01_Equipement_Library/Transfo/FB_Transfo_Base.TcPOU
FUNCTION_BLOCK FB_Transfo_Base
//////////////////
// High Voltage transformer with Transfo or DMCR detection . 
//////////////////

VAR_INPUT PERSISTENT
	// Parameters of the Object (instance/model specific) 

END_VAR

VAR_OUTPUT
	//Child objects
	
END_VAR

VAR_INPUT
		// Transfo

END_VAR

VAR
	///MesDataExd					: Transfo ; 
		MesCP_Read					: BOOL := TRUE;	(* Read function enable *)
		MesCP_Write					: BOOL := TRUE;	(* Write function enable *)	
END_VAR

METHOD M_AlarmManagement
//////////////////
// Manages High Voltage Transformer Alarms
/////////////////

VAR 
	// Method local variables (reinitialized at each cycle) 
	FB_AlarmCodeManager : FB_AlarmCodeManager ; 

	
END_VAR
END_METHOD

METHOD M_Execute
//////////////////
//  Method Calls 
/////////////////

VAR 
	// Method local variables (reinitialized at each cycle) 

END_VAR

	
// METHODS CALLS //
	M_Read();
	M_AlarmManagement();
END_METHOD

METHOD M_Read : BOOL
VAR_INPUT
END_VAR

VAR
	MesAuxTransfoGazDischarge: INT;
	MesAuxTransfoTempTrigger: INT;
END_VAR
END_METHOD

END_FUNCTION_BLOCK

// ---- 01_Equipement_Library/Transfo/FB_Transfo_HVCom.TcPOU
FUNCTION_BLOCK FB_Transfo_HVCom EXTENDS FB_Transfo_Base
//////////////////
// High Voltage transformer with Transfo or DMCR detection . 
//////////////////

VAR_INPUT PERSISTENT
	// Parameters of the Object (instance/model specific) 
	
END_VAR

VAR_OUTPUT
	//Child objects
	
END_VAR

VAR_INPUT

END_VAR

VAR
MesDataExd		AT %Q*			: Transfo_HV ; 
		
END_VAR

METHOD M_AlarmManagement
//////////////////
// Manages High Voltage Transformer Alarms
/////////////////

VAR 
	// Method local variables (reinitialized at each cycle) 
	FB_AlarmCodeManager : FB_AlarmCodeManager ; 

	
END_VAR



// ALARM CODE //
	FB_AlarmCodeManager(
		bAlarm1			:= MesDataExd.MesData.MesAlarmTemp ,				// Temperature Alarm
		bAlarm2			:= MesDataExd.MesData.MesAlarmGas  , 				// Gas Alarm
		bAlarm3			:= MesDataExd.MesData.MesAlarmOilLevel  , 			// Pressure Alarm
		bAlarm4			:= FALSE, 								//
		bAlarm5			:= FALSE, 								//
		bAlarm6			:= FALSE,                               //
		bAlarm7			:= FALSE,                               //
		bAlarm8			:= FALSE,                               //
		bAlarm9			:= FALSE, 								//
		bAlarm10		:= FALSE,                               //
		bAlarm11		:= FALSE,                               //
		bAlarm12		:= FALSE,                               //
		bAlarm13		:= FALSE, 								//
		bAlarm14		:= FALSE,                               //
		bAlarm15		:= FALSE , 								//      
		wAlarmCode		=>MesDataExd.MesData.MesAlarmCode);               

// WARNING CODE //
	FB_AlarmCodeManager(
		bAlarm1 		:= FALSE,   							//
		bAlarm2			:= FALSE, 		                   	 	//
		bAlarm3			:= FALSE, 		                      	//
		bAlarm4			:= FALSE, 		                    	//
		bAlarm5			:= FALSE,                               //
		bAlarm6			:= FALSE,                               //
		bAlarm7			:= FALSE,                               //
		bAlarm8			:= FALSE,                               //
		bAlarm9			:= FALSE,                               //
		bAlarm10		:= FALSE,                               //
		bAlarm11		:= FALSE,                               //
		bAlarm12		:= FALSE,                               //
		bAlarm13		:= FALSE,                               //
		bAlarm14		:= FALSE,                               //
		bAlarm15		:= FALSE,                               //
		wAlarmCode		=>MesDataExd.MesData.MesWarningCode);
		
// EVENT CODE //
	FB_AlarmCodeManager(
		bAlarm1			:= FALSE, 			// 
		bAlarm2			:= FALSE, 			// 
		bAlarm3			:= FALSE, 			// 
		bAlarm4			:= FALSE, 			// 
		bAlarm5			:= FALSE,         	//
		bAlarm6			:= FALSE,         	//
		bAlarm7			:= FALSE,         	//
		bAlarm8			:= FALSE,         	//
		bAlarm9			:= FALSE,         	//
		bAlarm10		:= FALSE,         	//
		bAlarm11		:= FALSE,         	//
		bAlarm12		:= FALSE,         	//
		bAlarm13		:= FALSE,         	//
		bAlarm14		:= FALSE,         	//
		bAlarm15		:= FALSE,         	//
		wAlarmCode		=>MesDataExd.MesData.MesEventCode);
END_METHOD

METHOD M_Read : BOOL
VAR_INPUT
END_VAR

VAR
	MesAuxTransfoGazDischarge: INT;
	MesAuxTransfoTempTrigger: INT;
END_VAR
END_METHOD

END_FUNCTION_BLOCK

// ---- 01_Equipement_Library/Transfo/FB_Transfo_MVCom.TcPOU
FUNCTION_BLOCK FB_Transfo_MVCom EXTENDS FB_Transfo_Base

//////////////////
// High Voltage transformer with Transfo or DMCR detection 
//////////////////

VAR_INPUT PERSISTENT
	// Parameters of the Object (instance/model specific) 
	
END_VAR

VAR_OUTPUT
	//Child objects
	
END_VAR

VAR_INPUT

	
END_VAR

VAR
MesDataExd	AT %Q*				: Transfo_MV ; 
		
END_VAR

METHOD M_AlarmManagement
//////////////////
// Manages High Voltage Transformer Alarms
/////////////////

VAR 
	// Method local variables (reinitialized at each cycle) 
	FB_AlarmCodeManager : FB_AlarmCodeManager ; 

	
END_VAR
// ALARM CODE //
	FB_AlarmCodeManager(
		bAlarm1			:= MesDataExd.MesData.MesAlarmTemp  ,				// Temperature Alarm
		bAlarm2			:= MesDataExd.MesData.MesAlarmGas  , 				// Gas Alarm
		bAlarm3			:= MesDataExd.MesData.MesAlarmOilLevel  , 			// Oil Level Alarm
		bAlarm4			:= FALSE, 								//
		bAlarm5			:= FALSE, 								//
		bAlarm6			:= FALSE,                               //
		bAlarm7			:= FALSE,                               //
		bAlarm8			:= FALSE,                               //
		bAlarm9			:= FALSE, 								//
		bAlarm10		:= FALSE,                               //
		bAlarm11		:= FALSE,                               //
		bAlarm12		:= FALSE,                               //
		bAlarm13		:= FALSE, 								//
		bAlarm14		:= FALSE,                               //
		bAlarm15		:= FALSE , 								//      
		wAlarmCode		=>MesDataExd.MesData.MesAlarmCode);               

// WARNING CODE //
	FB_AlarmCodeManager(
		bAlarm1 		:= FALSE,   							//
		bAlarm2			:= FALSE, 		                   	 	//
		bAlarm3			:= FALSE, 		                      	//
		bAlarm4			:= FALSE, 		                    	//
		bAlarm5			:= FALSE,                               //
		bAlarm6			:= FALSE,                               //
		bAlarm7			:= FALSE,                               //
		bAlarm8			:= FALSE,                               //
		bAlarm9			:= FALSE,                               //
		bAlarm10		:= FALSE,                               //
		bAlarm11		:= FALSE,                               //
		bAlarm12		:= FALSE,                               //
		bAlarm13		:= FALSE,                               //
		bAlarm14		:= FALSE,                               //
		bAlarm15		:= FALSE,                               //
		wAlarmCode		=>MesDataExd.MesData.MesWarningCode);
		
// EVENT CODE //
	FB_AlarmCodeManager(
		bAlarm1			:= FALSE, 			// 
		bAlarm2			:= FALSE, 			// 
		bAlarm3			:= FALSE, 			// 
		bAlarm4			:= FALSE, 			// 
		bAlarm5			:= FALSE,         	//
		bAlarm6			:= FALSE,         	//
		bAlarm7			:= FALSE,         	//
		bAlarm8			:= FALSE,         	//
		bAlarm9			:= FALSE,         	//
		bAlarm10		:= FALSE,         	//
		bAlarm11		:= FALSE,         	//
		bAlarm12		:= FALSE,         	//
		bAlarm13		:= FALSE,         	//
		bAlarm14		:= FALSE,         	//
		bAlarm15		:= FALSE,         	//
		wAlarmCode		=>MesDataExd.MesData.MesEventCode);
END_METHOD

METHOD M_Read : BOOL
VAR_INPUT
END_VAR

VAR
	MesAuxTransfoGazDischarge: INT;
	MesAuxTransfoTempTrigger: INT;
END_VAR
END_METHOD

END_FUNCTION_BLOCK

// ---- 01_Equipement_Library/Transfo/FB_Transfo_MV.TcPOU
FUNCTION_BLOCK FB_Transfo_MV EXTENDS FB_Transfo_Base
//////////////////
// High Voltage transformer with DGPT2 detection . 
//////////////////

VAR_INPUT PERSISTENT
	// Parameters of the Object (instance/model specific) 
	ParamNC					: BOOL  ; 			(* Normally closed inputs . If TRUE , 1 =  no alarms. *)
END_VAR

VAR_OUTPUT
	//Child objects
	
END_VAR

VAR_INPUT
		// Transfo
	IN_MesWarningTemp_IO				: BOOL ; 		// (NA) Warning Oil Temperature IO
	IN_MesAlarmTemp_IO					: BOOL ; 		// (NA) Alarm Oil Temperature   IO
	IN_MesAlarmGas_IO					: BOOL ; 		// (NA) Gas Alarm               IO
	IN_MesAlarmPressure_IO				: BOOL ; 		// (NA) Oil Pressure Alarm		IO
	IN_MesAlarmsSynthesis_IO			: BOOL ;        // (NA) Alarms synthesis        IO 
	IN_MesAlarmOilLevel_IO				: BOOL ;		// (NA) Alarm oil level			IO
END_VAR

VAR
	MesDataExd				   : Transfo_MV ; 
	
END_VAR

METHOD M_AlarmManagement
//////////////////
// Manages High Voltage Transformer Alarms
/////////////////

VAR 
	// Method local variables (reinitialized at each cycle) 
	FB_AlarmCodeManager : FB_AlarmCodeManager ; 

	
END_VAR
IF ParamNC THEN 
	MesDataExd.MesData.MesAlarmsSynthesis		:= NOT IN_MesAlarmsSynthesis_IO ; 
	MesDataExd.MesData.MesAlarmGas				:= NOT IN_MesAlarmGas_IO ; 
	MesDataExd.MesData.MesAlarmOilLevel 		:= NOT IN_MesAlarmOilLevel_IO ; 
	MesDataExd.MesData.MesAlarmTemp				:= NOT IN_MesAlarmTemp_IO ;  
	MesDataExd.MesData.MesWarningTemp			:= NOT  IN_MesWarningTemp_IO ; 
ELSE
	MesDataExd.MesData.MesAlarmsSynthesis		:= IN_MesAlarmsSynthesis_IO ; 
	MesDataExd.MesData.MesAlarmGas				:= IN_MesAlarmGas_IO ; 
	MesDataExd.MesData.MesAlarmOilLevel 		:= IN_MesAlarmOilLevel_IO ; 
	MesDataExd.MesData.MesAlarmTemp				:= IN_MesAlarmTemp_IO ;  
	MesDataExd.MesData.MesWarningTemp			:=  IN_MesWarningTemp_IO ; 

END_IF



// ALARM CODE //
	FB_AlarmCodeManager(
		bAlarm1			:= MesDataExd.MesData.MesAlarmTemp ,				// Temperature Alarm
		bAlarm2			:= MesDataExd.MesData.MesAlarmGas  , 				// Gas Alarm
		bAlarm3			:= MesDataExd.MesData.MesAlarmOilLevel  , 			// Pressure Alarm
		bAlarm4			:= MesDataExd.MesData.MesAlarmsSynthesis, 			// Alarms Synthesis Gaz,Pressure,T
		bAlarm5			:= FALSE ,//                
		bAlarm6			:= FALSE ,//               
		bAlarm7			:= FALSE ,//            
		bAlarm8			:= FALSE ,//
		bAlarm9			:= FALSE, 								//
		bAlarm10		:= FALSE,                               //
		bAlarm11		:= FALSE,                               //
		bAlarm12		:= FALSE,                               //
		bAlarm13		:= FALSE, 								//
		bAlarm14		:= FALSE,                               //
		bAlarm15		:= FALSE , 								//      
		wAlarmCode		=>MesDataExd.MesData.MesAlarmCode);               

// WARNING CODE //
	FB_AlarmCodeManager(
		bAlarm1 		:= MesDataExd.MesData.MesWarningTemp,   			// Temperature Warning
		bAlarm2			:= FALSE ,//
		bAlarm3			:= FALSE, 		                      	//
		bAlarm4			:= FALSE, 		                    	//
		bAlarm5			:= FALSE,                               //
		bAlarm6			:= FALSE,                               //
		bAlarm7			:= FALSE,                               //
		bAlarm8			:= FALSE,                               //
		bAlarm9			:= FALSE,                               //
		bAlarm10		:= FALSE,                               //
		bAlarm11		:= FALSE,                               //
		bAlarm12		:= FALSE,                               //
		bAlarm13		:= FALSE,                               //
		bAlarm14		:= FALSE,                               //
		bAlarm15		:= FALSE,                               //
		wAlarmCode		=>MesDataExd.MesData.MesWarningCode);
		
// EVENT CODE //
	FB_AlarmCodeManager(
		bAlarm1			:= NOT MesDataExd.MesData.MesAlarmTemp ,			// Temperature Alarm back to normal       
		bAlarm2			:= NOT MesDataExd.MesData.MesAlarmGas  , 			// Gas Alarm back to normal              
		bAlarm3			:= NOT MesDataExd.MesData.MesAlarmOilLevel  , 		// Pressure Alarm back to normal     
		bAlarm4			:= NOT MesDataExd.MesData.MesAlarmsSynthesis, 		// No alarms active                  
		bAlarm5			:= NOT MesDataExd.MesData.MesWarningTemp,   		// Temperature Warning End
		bAlarm6			:= FALSE ,				//
		bAlarm7			:= FALSE,         	//
		bAlarm8			:= FALSE,         	//
		bAlarm9			:= FALSE,         	//
		bAlarm10		:= FALSE,         	//
		bAlarm11		:= FALSE,         	//
		bAlarm12		:= FALSE,         	//
		bAlarm13		:= FALSE,         	//
		bAlarm14		:= FALSE,         	//
		bAlarm15		:= FALSE,         	//
		wAlarmCode		=>MesDataExd.MesData.MesEventCode);
END_METHOD

END_FUNCTION_BLOCK

// ---- 01_Equipement_Library/UPS/FB_UPS_PS10048.TcPOU
FUNCTION_BLOCK FB_UPS_PS10048 EXTENDS FB_UPS_Base
//////////////////
// SEPAM system for High Voltage or Low Voltage Grid Protection. 
//////////////////

VAR_INPUT 
	ParamTcpPort				: UINT:=502;		(* (NA) Tcp port *)
	ParamIPAddress				: STRING;           (* (NA) IP address*)
	ParamUnitID					: BYTE;             (* (NA) Unit ID*)
END_VAR

VAR_OUTPUT
	
END_VAR

VAR_INPUT

END_VAR

VAR
MesDataExd    	AT %Q*	: UPS_PS10048;
	FB_ModbusRead	          	: ARRAY[1..4] OF FB_ModbusRead; 
			
	MesBlock1_Temp 				: ARRAY [1..1] OF WORD ; 
	MesBlock2_Temp 				: ARRAY [1..11] OF WORD ; 
	MesBlock3_Temp 				: ARRAY [1..8] OF WORD ; 
	MesBlock4_Temp 				: ARRAY [1..2] OF WORD ; 
	
	AX_ModbusReadAlarm			: ARRAY[1..4] OF BOOL;
	AX_ModbusReadAlarmId		: ARRAY[1..4] OF UDINT;	
END_VAR

METHOD M_AlarmManagement
//////////////////
// Manages Sepam Alarms. Alarms opens HT CB until Sepam manual Reset. Warning Opens CB-L but does not maintain warning.
/////////////////

VAR 
	// Method local variables (reinitialized at each cycle) 
	FB_AlarmCodeManager 	: FB_AlarmCodeManager; 
 	ComWarning				: BOOL;
	ComAlarms				: BOOL;
END_VAR
// ALARM CODE //
	FB_AlarmCodeManager(
		bAlarm1			:= MesDataExd.MesData.MesAlarmCom,			// Com alarm
		bAlarm2			:= MesDataExd.MesData.MesFault_Major,				// True := Major fault : cannot recover
		bAlarm3			:= MesDataExd.MesData.MesAlarm_AcOff,				// True := AC off		
		bAlarm4			:= MesDataExd.MesData.MesAlarm_GeneralOff,			// True := Imminent shut down
		bAlarm5			:= MesDataExd.MesData.MesFault_Bat,					// True := Battery disconnected
		bAlarm6			:= MesDataExd.MesData.MesFault_Charger,				// True := Charger out of order										 
		bAlarm7			:= MesDataExd.MesData.MesFault_12V,					// True := 12V absent 
		bAlarm8			:= MesDataExd.MesData.MesFault_48V,					// True := 48V absent
		bAlarm9			:= MesDataExd.MesData.MesToggleRead,				// True := AC power supply low 
		bAlarm10		:= FALSE, 									//										
		bAlarm11		:= FALSE,                                   //
		bAlarm12		:= FALSE,                                   //
		bAlarm13		:= FALSE,                                   //
		bAlarm14		:= FALSE,                                   //
		bAlarm15		:= FALSE, 									// 
		wAlarmCode		=>MesDataExd.MesData.MesAlarmCode);		

// WARNING CODE //
	FB_AlarmCodeManager(
		bAlarm1			:= MesDataExd.MesData.MesFault_Minor,				// True := Minor fault (overtemp, overcurrent, overvolt)
		bAlarm2			:= MesDataExd.MesData.MesAlarm_Ulow ,		// Battery  Capacity is low 
		bAlarm4			:= FALSE,									//
		bAlarm5			:= FALSE,									//
		bAlarm6			:= FALSE,									//
		bAlarm7			:= FALSE,									// 
		bAlarm8			:= FALSE,									// 
		bAlarm9			:= FALSE,									// 
		bAlarm10		:= FALSE,									// 
		bAlarm11		:= FALSE,									// 
		bAlarm12		:= FALSE,									// 
		bAlarm13		:= FALSE,									// 
		bAlarm14		:= FALSE,									// 
		bAlarm15		:= FALSE,									// 
		wAlarmCode		=>MesDataExd.MesData.MesWarningCode);					

// EVENT CODE //
	FB_AlarmCodeManager(
		bAlarm1			:=FALSE, 									// 
		bAlarm2			:=FALSE, 									// 
		bAlarm3			:=FALSE, 									// 
		bAlarm4			:=FALSE, 									// 
		bAlarm5			:=FALSE, 									//
		bAlarm6			:=FALSE,        							//
		bAlarm7			:=FALSE,        							//
		bAlarm8			:=FALSE,        							//
		bAlarm9			:=FALSE,        							//
		bAlarm10		:=FALSE, 									//
		bAlarm11		:=FALSE,        							//
		bAlarm12		:=FALSE,        							//
		bAlarm13		:=FALSE,        							//
		bAlarm14		:=FALSE,        							//
		bAlarm15		:=FALSE, 									//
		wAlarmCode		= MesDataExd.MesData.MesEventCode);					
		
MesData := MesDataExd.MesData.
END_METHOD

METHOD M_Evaluate
VAR_INPUT
END_VAR

VAR
END_VAR
END_METHOD

METHOD M_Read
//////////////////
//  Method Calls 
/////////////////

VAR_INPUT
	
END_VAR
VAR 
	MW					: FB_MergeWordsToFloat;
	MW_1				: FB_MergeWordsToDint;
END_VAR
// CP-Read / Write 

MesDataExd.MesData.MesCP_Read := MesCP_Read ; 

IF MesCP_Read  THEN		
	
	FB_ModbusRead[1]
		(
			nTCPPort		:= ParamTcpPort,
			ClockRead		:= MesCP_Read AND ClockRead, 
			Reset			:= CmdClearFault_G OR IN_CmdReset_L,
			sIPAddr			:= ParamIPAddress ,
			nUnitID			:= 1, 
			tTimeout		:= T#5S,
			nQuantity		:= 1, 
			nMBAddr			:= 44000 , 
			cbLength		:= SIZEOF(MesBlock1_Temp) , 
			pDestAddr		:= ADR(MesBlock1_Temp) , 
			ModbusReadAlarm	=> AX_ModbusReadAlarm[1] , 
			ErrorId			=> AX_ModbusReadAlarmId[1]
		);
		
	FB_ModbusRead[2]
		(
			nTCPPort		:= ParamTcpPort,
			ClockRead		:= MesCP_Read AND ClockRead, 
			Reset			:= CmdClearFault_G OR IN_CmdReset_L,
			sIPAddr			:= ParamIPAddress ,
			nUnitID			:= 1, 
			tTimeout		:= T#5S,
			nQuantity		:= 9, 
			nMBAddr			:= 44100 , 
			cbLength		:= SIZEOF(MesBlock2_Temp) , 
			pDestAddr		:= ADR(MesBlock2_Temp) , 
			ModbusReadAlarm	=> AX_ModbusReadAlarm[2], 
			ErrorId			=> AX_ModbusReadAlarmId[2]
		);
		
		FB_ModbusRead[3]
		(
			nTCPPort		:= ParamTcpPort,
			ClockRead		:= MesCP_Read AND ClockRead	, 
			Reset			:= CmdClearFault_G OR IN_CmdReset_L,
			sIPAddr			:= ParamIPAddress ,
			nUnitID			:= 1, 
			tTimeout		:= T#5S,
			nQuantity		:= 6, 
			nMBAddr			:= 44150 , 
			cbLength		:= SIZEOF(MesBlock3_Temp) , 
			pDestAddr		:= ADR(MesBlock3_Temp) , 
			ModbusReadAlarm	=> AX_ModbusReadAlarm[3], 
			ErrorId			=> AX_ModbusReadAlarmId[3]
		);
	
			FB_ModbusRead[4]
		(
			nTCPPort		:= ParamTcpPort,
			ClockRead		:= MesCP_Read AND ClockRead, 
			Reset			:= CmdClearFault_G OR IN_CmdReset_L,
			sIPAddr			:= ParamIPAddress,
			nUnitID			:= 1, 
			tTimeout		:= T#5S,
			nQuantity		:= 2, 
			nMBAddr			:= 44050 , 
			cbLength		:= SIZEOF(MesBlock4_Temp) , 
			pDestAddr		:= ADR(MesBlock4_Temp) , 
			ModbusReadAlarm	=> AX_ModbusReadAlarm[4], 
			ErrorId			=> AX_ModbusReadAlarmId[4]
		);
		
		//COM
	MesDataExd.MesData.MesAlarmCom 			:= NOT WORD_TO_BOOL(MesBlock1_Temp[1]);
	MesDataExd.MesSoc						:= WORD_TO_REAL(MesBlock2_Temp[1])* 0.01;
		
		MW( WORD_STRONG:= MesBlock2_Temp[3  ],	WORD_WEAK := MesBlock2_Temp[2  ], VAR_OUT := MesDataExd.MesSoc);
		MW( WORD_STRONG:= MesBlock2_Temp[5  ],	WORD_WEAK := MesBlock2_Temp[4  ], VAR_OUT := MesDataExd.MesUdc_48V);
		MW( WORD_STRONG:= MesBlock2_Temp[7  ],	WORD_WEAK := MesBlock2_Temp[6  ], VAR_OUT := MesDataExd.MesUdc_12V);
		MW( WORD_STRONG:= MesBlock2_Temp[9  ],	WORD_WEAK := MesBlock2_Temp[8  ], VAR_OUT := MesDataExd.MesUBatt);
		MW( WORD_STRONG:= MesBlock2_Temp[11 ],	WORD_WEAK := MesBlock2_Temp[10 ], VAR_OUT := MesDataExd.MesIdc_Bat);
	
		MW( WORD_STRONG:= MesBlock3_Temp[2  ],	WORD_WEAK := MesBlock3_Temp[1  ], VAR_OUT := MesDataExd.MesDischarge);
	MesDataExd.MesEbackUp		  		:= WORD_TO_REAL(MesBlock3_Temp[3  ]) * 0.01;
	MesDataExd.MesEBackUpEna	  		:= WORD_TO_BOOL(MesBlock3_Temp[4  ]);
	MesDataExd.MesBatTestPer	  		:= WORD_TO_BOOL(MesBlock3_Temp[5  ]);
	MesDataExd.MesVacTripSelect	  		:= WORD_TO_BOOL(MesBlock3_Temp[6  ]);	
		MW( WORD_STRONG:= MesBlock3_Temp[8  ],	WORD_WEAK := MesBlock3_Temp[7  ], VAR_OUT := MesDataExd.MesCapacity_Nom);
		
		MesDataExd.MesFault_Minor 			:= MesBlock4_Temp[1].8;
		MesDataExd.MesFault_Major  		:= MesBlock4_Temp[1].11;
		MesDataExd.MesAlarm_AcOff 			:= MesBlock4_Temp[2].0;
		MesDataExd.MesAlarm_GeneralOff		:= MesBlock4_Temp[2].1;
		MesDataExd.MesData.MesAlarm_Ulow	:= MesBlock4_Temp[2].2;
		MesDataExd.MesFault_Bat			:= MesBlock4_Temp[2].3;
//		MesDataExd.MesFault_Bat			:= MesBlock4_Temp[2].4;
		MesDataExd.MesFault_12V			:= MesBlock4_Temp[2].5;
		MesDataExd.MesFault_48V			:= MesBlock4_Temp[2].6;
		MesDataExd.MesAlarm_AcLow			:= MesBlock4_Temp[2].7; 
		
END_IF 

	// properties update 
MesDataExd.MesData.MesUdc 				:= MesDataExd.MesUdc_12V ; 
MesDataExd.MesData.MesDischarging 		:= MesDataExd.MesAlarm_AcOff 	; 
	
MesDataExd.MesData.MesAlarmState 		:= MesDataExd.MesFault_Minor OR MesDataExd.MesFault_Major OR MesDataExd.MesAlarm_GeneralOff OR 
											 MesDataExd.MesFault_Bat OR MesDataExd.MesFault_Bat  ;
END_METHOD

END_FUNCTION_BLOCK

// ---- 01_Equipement_Library/UPS/FB_UPS_Base.TcPOU
FUNCTION_BLOCK FB_UPS_Base
//////////////////
// UPS 
//////////////////
VAR_INPUT PERSISTENT
	// Parameters of the Object (instance/model specific) 
		ParamTimeOut					: TIME := T#2S;		(* (s) Modbus Timeout*)
		ParamClockReadTime				: TIME := T#1S;		(* (s) Modbus Reading Frequency *)
		ParamNC							: BOOL := FALSE; 	(* (NA)False: TRUE = Closed, True : TRUE = opened*)
		                                
		ParamTempoComAlarm				: TIME := T#2S;		(* (s) Tempo before raising a communication alarm*)
		ParamTempoComWarning			: TIME := T#1S;		(* (s) Tempo before raising a communication warning*)
		ParamTP_Impulsion				: TIME := T#5S;		(* (s) TP Impulsion = 5s *)
END_VAR                                 
                                        
VAR_OUTPUT                              
	//Child objects                     
		OUT_CmdRelance_IO				: BOOL;
END_VAR                                 
                                        
VAR_INPUT                               
	// I/O Inputs                       
		IN_MesDischarging_IO		  	: BOOL;
		IN_MesBatLow_IO		   			: BOOL;
		IN_MesFault_IO					: BOOL;

		IN_CmdReStartUPS				: BOOL;
		
		IN_CmdToggleRead				: BOOL;
		IN_CmdReset_L					: BOOL; 
END_VAR

VAR
	//M_ALARMMANAGEMENT VARIABLES//
		TON_ComAlarm					: TON;
		TON_ComWarning					: TON;	

		MesWarningCom					: BOOL ; 			// (NA) [P,H] True if bad modbus communication 
			
	//M_READ//
//	MesDataExd					: UPS ; 

	//M_EXECUTE //
		TP1								: TP;
		ClockRead			AT %Q*		: BOOL;
   		
    //M_CP VARIABLES//
		Trig_Cmd_Read					: R_TRIG;                                                                                        
                                                                                       
		CmdRelanceChargeur				: BOOL;
		CP_Relance						: BOOL;
		TP_Relance						: TP;
		MesCP_Read					: BOOL := TRUE;	(* Read function enable *)
		MesCP_Write					: BOOL := TRUE;	(* Write function enable *)   
END_VAR

METHOD M_AlarmManagement
//////////////////
// Manages Sepam Alarms. Alarms opens HT CB until Sepam manual Reset . Warning Opens CB-L but does not maintain warning
/////////////////

VAR 
	// Method local variables (reinitialized at each cycle) 
	FB_AlarmCodeManager 	: FB_AlarmCodeManager ; 

 
END_VAR
END_METHOD

METHOD M_Execute
//////////////////
//  Method Calls 
/////////////////

VAR 
	// Method local variables (reinitialized at each cycle) 

END_VAR


// METHODS CALLS // 
Trig_Cmd_Read(CLK:=IN_CmdToggleRead);
CP_Relance	:= IN_CmdReStartUPS ; 	
IF Trig_Cmd_Read.Q THEN
	//IN_CmdToggleRead := FALSE;
	MesCP_Read := NOT MesCP_Read;
	
END_IF

	TP1(IN:=NOT TP1.Q , PT:= ParamClockReadTime);
	ClockRead 		:= TP1.Q;

	TP_Relance(IN:= CP_Relance , PT:=ParamTP_Impulsion) ;
	OUT_CmdRelance_IO	 := TP_Relance.Q ;
	
	M_Read(); 
	M_AlarmManagement() ;
END_METHOD

METHOD M_Read
//////////////////
//  Read Modbus Variable for PCS . 
/////////////////
VAR 
	// Method local variables (reinitialized at each cycle) 
		

END_VAR
END_METHOD

END_FUNCTION_BLOCK

// ---- 01_Equipement_Library/UPS/FB_UPS_CXC.TcPOU
FUNCTION_BLOCK FB_UPS_CXC EXTENDS FB_UPS_Base
//////////////////
// UPS 
//////////////////
VAR_INPUT PERSISTENT
	// Parameters of the Object (instance/model specific) 

		{attribute 'OPC.UA.DA' := '1'} 
		ParamIPAddress				: STRING 	:= '192.168.20.66'; 	// (NA)Config: IP Adress of PV INverter
		{attribute 'OPC.UA.DA' := '1'} 
		ParamUnitID 				: BYTE  	:= 1; 			  		// (NA)   Modbus Unit ID. 
		{attribute 'OPC.UA.DA' := '1'} 
		ParamTCPPort				: UINT		:= 502;					// (NA) TCP port for modbus
		
END_VAR

VAR_OUTPUT
	//Child objects
	
END_VAR

VAR_INPUT
	// I/O Inputs
		IN_MesCbUPS_IO					: BOOL ; // 1 = opened. 
END_VAR

VAR
	//M_ALARMMANAGEMENT VARIABLES//

	//M_READ//
		MesDataExd						AT %Q*	: UPS_CXC ; 
		AX_ModbusRead		   		: ARRAY [1..2] OF FB_ModbusRead ; 					// (NA) FB for Modbus Reading
		ModbusReadInput				: FB_ModbusReadInput ; 		       
                                 
		MesBlock_Temp 				: ARRAY [1..2] OF ARRAY[1..120]  OF WORD; 			// (NA) Temporary Block with multiple modbus reading (Caution : Double Word variables)
		MesBlockInput				: ARRAY[1..1] OF BYTE ; 
		
	
	//M_EXECUTE //

		
END_VAR

METHOD M_AlarmManagement
//////////////////
// Manages Sepam Alarms. Alarms opens HT CB until Sepam manual Reset . Warning Opens CB-L but does not maintain warning
/////////////////

VAR 
	// Method local variables (reinitialized at each cycle) 
	FB_AlarmCodeManager 	: FB_AlarmCodeManager ; 

 
END_VAR
	//Alarm
	
	TON_ComAlarm	(IN:= (AX_ModbusRead[1].ModbusReadAlarm) AND (AX_ModbusRead[2].ModbusReadAlarm) AND (ModbusReadInput.ModbusReadAlarm) , PT:= ParamTempoComAlarm, 	Q=>MesDataExd.MesData.MesAlarmCom) ;	
	TON_ComWarning	(IN:= (AX_ModbusRead[1].ModbusReadAlarm) OR  (AX_ModbusRead[2].ModbusReadAlarm) OR  (ModbusReadInput.ModbusReadAlarm) , PT:= ParamTempoComWarning, 	Q=>MesWarningCom) ;	


// ALARM CODE //
	FB_AlarmCodeManager(
		bAlarm1				:= FALSE , 				 									//  
		bAlarm2				:= MesDataExd.MesData.MesAlarm_Ulow ,						// Battery SoC is low
		bAlarm3				:= MesDataExd.MesData.MesAlarmState ,					// UPS Fault synthesis
		bAlarm4				:= MesDataExd.MesOverTempBatt,     							// Battery overtemperature
		bAlarm5				:= FALSE,         											// 
		bAlarm6				:= FALSE, 													//
		bAlarm7				:= FALSE, 													//
		bAlarm8				:= FALSE,                                                   //
		bAlarm9				:= FALSE,                                                   //
		bAlarm10			:= FALSE,                                                   //
		bAlarm11			:= FALSE,                                                   //
		bAlarm12			:= FALSE,                                                   //
		bAlarm13			:= FALSE,                                                   //
		bAlarm14			:= FALSE,                                                   //
		bAlarm15			:= FALSE , 													//
		wAlarmCode			=> MesDataExd.MesData.MesAlarmCode);

// WARNING CODE //
	FB_AlarmCodeManager(
		bAlarm1			:= MesDataExd.MesData.MesDischarging , 				 			// UPS is discharging  , 														// 
		bAlarm2			:= MesDataExd.MesCBUpsOpened, 									// CB UPS Opened . 
		bAlarm3			:= MesWarningCom, 												// Communication warning  #COM
		bAlarm4			:= MesDataExd.MesData.MesAlarmCom,         						// Communication alarm, 	#COM													// 
		bAlarm5			:= FALSE, 														//
		bAlarm6			:= FALSE,                                                       //
		bAlarm7			:= FALSE,                                                       //
		bAlarm8			:= FALSE,                                                       //
		bAlarm9			:= FALSE,                                                       //
		bAlarm10		:= FALSE,                                                       //
		bAlarm11		:= FALSE,                                                       //
		bAlarm12		:= FALSE,                                                       //
		bAlarm13		:= FALSE,                                                       //
		bAlarm14		:= FALSE,                                                       //
		bAlarm15		:= FALSE,                                                       //
		wAlarmCode		=> MesDataExd.MesData.MesWarningCode);

// EVENT CODE //
	FB_AlarmCodeManager(
		bAlarm1			:=FALSE, 													// 
		bAlarm2			:=FALSE, 													// 
		bAlarm3			:=FALSE, 													// 
		bAlarm4			:=FALSE, 													// 
		bAlarm5			:=FALSE, 													//
		bAlarm6			:=FALSE,        											//
		bAlarm7			:=FALSE,        											//
		bAlarm8			:=FALSE,        											//
		bAlarm9			:=FALSE,        											//
		bAlarm10		:=FALSE,        											//
		bAlarm11		:=FALSE,        											//
		bAlarm12		:=FALSE,        											//
		bAlarm13		:=FALSE,        											//
		bAlarm14		:=FALSE,        											//
		bAlarm15		:=FALSE,        											//
		wAlarmCode		=> MesDataExd.MesData.MesEventCode);
END_METHOD

METHOD M_Read
//////////////////
//  Read Modbus Variable for PCS . 
/////////////////
VAR 
	// Method local variables (reinitialized at each cycle) 
		
		AX_Addr				: ARRAY[1..3] OF UINT := [16#82, 		16#C2, 	16#101];
		AX_Qty				: ARRAY[1..3] OF UINT := [16, 		6, 	4];
		
		MW 					: FB_MergeWordsToDint; 
END_VAR
// CP-Read / Write 

MesDataExd.MesData.MesCP_Read := MesCP_Read ; 

IF MesCP_Read  THEN	

AX_ModbusRead[1]
(
	pDestAddr 		:= ADR(MesBlock_Temp[1]),
	sIPAddr 		:= ParamIPAddress,
	tTimeout 		:= ParamTimeout,
	nQuantity 		:= AX_Qty[1],
	ntcpport 		:= ParamTCPPort,
	nMBAddr 		:= AX_Addr[1]-2,
	nUnitID 		:= ParamUnitID,
	cbLength 		:= SIZEOF(MesBlock_Temp[1]),
	ClockRead 		:= ClockRead AND MesCP_Read,
	Reset 			:= CmdClearFault_G OR IN_CmdReset_L,
);


AX_ModbusRead[2]
(
	pDestAddr 		:= ADR(MesBlock_Temp[2]),
	sIPAddr 		:= ParamIPAddress,
	tTimeout 		:= ParamTimeout,
	nQuantity 		:= AX_Qty[2],
	ntcpport 		:= ParamTCPPort,
	nMBAddr 		:= AX_Addr[2]-2,
	nUnitID 		:= ParamUnitID,
	cbLength 		:= SIZEOF(MesBlock_Temp[2]),
	ClockRead 		:= ClockRead AND MesCP_Read,
	Reset 			:= CmdClearFault_G OR IN_CmdReset_L
);


ModbusReadInput
(
	pDestAddr 		:= ADR(MesBlockInput),
	sIPAddr 		:= ParamIPAddress,
	tTimeout 		:= ParamTimeout,
	nQuantity 		:= AX_Qty[3],
	ntcpport 		:= ParamTCPPort,
	nMBAddr 		:= AX_Addr[3]-1,
	nUnitID 		:= ParamUnitID,
	cbLength 		:= SIZEOF(MesBlockInput),
	ClockRead 		:= ClockRead AND MesCP_Read,
	Reset 			:= GVL_CFG.CmdClearFault_G OR IN_CmdReset_L
);


	


MW(WORD_STRONG:= MesBlock_Temp[1][3], WORD_WEAK := MesBlock_Temp[1][4],SIGNED:=TRUE, FIX:=2 , SIZE:=2, VAR_OUT:=MesDataExd.MesIload);
MW(WORD_STRONG:= MesBlock_Temp[1][5], WORD_WEAK := MesBlock_Temp[1][6],SIGNED:=TRUE, FIX:=2 , SIZE:=2, VAR_OUT:=MesDataExd.MesUBatt);
MW(WORD_STRONG:= MesBlock_Temp[1][7], WORD_WEAK := MesBlock_Temp[1][8],SIGNED:=TRUE, FIX:=2 , SIZE:=2, VAR_OUT:=MesDataExd.MesIBatt);
MW(WORD_STRONG:= MesBlock_Temp[1][15], WORD_WEAK := MesBlock_Temp[1][16],SIGNED:=TRUE, FIX:=2 , SIZE:=2, VAR_OUT:=MesDataExd.MesSoC);

MW(WORD_STRONG:= MesBlock_Temp[2][1], WORD_WEAK := MesBlock_Temp[2][2],SIGNED:=TRUE, FIX:=2 , SIZE:=2, VAR_OUT:=MesDataExd.MesIdc);
MW(WORD_STRONG:= MesBlock_Temp[2][3], WORD_WEAK := MesBlock_Temp[2][4],SIGNED:=TRUE, FIX:=2 , SIZE:=2, VAR_OUT:=MesDataExd.MesData.MesUdc);
MW(WORD_STRONG:= MesBlock_Temp[2][5], WORD_WEAK := MesBlock_Temp[2][6],SIGNED:=TRUE, FIX:=2 , SIZE:=2, VAR_OUT:=MesDataExd.MesU);

MesDataExd.MesData.MesAlarm_Ulow := MesBlockInput[1].1	; // Low battery capacity 
MesDataExd.MesOverTempBatt	:= MesBlockInput[1].2 ; // OverTemp battery 
MesDataExd.MesData.MesDischarging := MesBlockInput[1].3 OR IN_MesDischarging_IO ; 
MesDataExd.MesData.MesAlarmState := IN_MesFault_IO ; 


END_IF


IF ParamNC THEN
	MesDataExd.MesCBUpsOpened := IN_MesCbUPS_IO ; 
	
ELSE 
 	MesDataExd.MesCBUpsOpened := NOT IN_MesCbUPS_IO ;
END_IF
END_METHOD

END_FUNCTION_BLOCK

// ---- 01_Equipement_Library/UPS/FB_UPS_Eneris.TcPOU
FUNCTION_BLOCK FB_UPS_ENERIS EXTENDS FB_UPS_Base
//////////////////
// UPS 
//////////////////
VAR_INPUT PERSISTENT
	// Parameters of the Object (instance/model specific) 
	
END_VAR

VAR_OUTPUT
	//Child objects
	
END_VAR

VAR_INPUT
	// I/O Inputs
		IN_MesCbUPS_IO					: BOOL ; // 1 = opened. 
END_VAR

VAR
	//M_ALARMMANAGEMENT VARIABLES//
		
	//M_READ//

	MesDataExd				: UPS_ENERIS ; 
	
		
	//M_EXECUTE //
		
	
END_VAR

METHOD M_AlarmManagement
//////////////////
// Manages Sepam Alarms. Alarms opens HT CB until Sepam manual Reset . Warning Opens CB-L but does not maintain warning
/////////////////

VAR 
	// Method local variables (reinitialized at each cycle) 
	FB_AlarmCodeManager 	: FB_AlarmCodeManager ; 

 
END_VAR
IF ParamNC THEN 
MesDataExd.MesData.MesDischarging  	:=  NOT IN_MesDischarging_IO;
MesDataExd.MesData.MesAlarm_Ulow 	 	:=  NOT IN_MesBatLow_IO;
MesDataExd.MesData.MesAlarmState 		:=  NOT IN_MesFault_IO;
	
ELSE
MesDataExd.MesData.MesDischarging  	:=  IN_MesDischarging_IO;
MesDataExd.MesData.MesAlarm_Ulow 	 	:=  IN_MesBatLow_IO;
MesDataExd.MesData.MesAlarmState 		:=  IN_MesFault_IO;

END_IF

// ALARM CODE //
	FB_AlarmCodeManager(
		bAlarm1				:= FALSE , 				 						// 
		bAlarm2				:= MesDataExd.MesData.MesAlarm_Ulow ,						// Battery SoC is low 
		bAlarm3				:= MesDataExd.MesData.MesAlarmState ,						// UPS Fault synthesis		
		bAlarm4				:= FALSE,     									// 
		bAlarm5				:= FALSE,         								//  
		bAlarm6				:= FALSE, 										// 
		bAlarm7				:= FALSE,                                       //
		bAlarm8				:= FALSE,                                       //
		bAlarm9				:= FALSE,                                       //
		bAlarm10			:= FALSE,                                       //
		bAlarm11			:= FALSE,                                       //
		bAlarm12			:= FALSE,                                       //
		bAlarm13			:= FALSE,                                       //
		bAlarm14			:= FALSE,                                       //
		bAlarm15			:= FALSE ,	 									//
		wAlarmCode			=>MesDataExd.MesData.MesAlarmCode);

// WARNING CODE //
	FB_AlarmCodeManager(
		bAlarm1			:= MesDataExd.MesData.MesDischarging , 				 		// UPS is discharging  		
		bAlarm2			:= FALSE, 											// 
		bAlarm3			:= FALSE, 											// 
		bAlarm4			:= FALSE, 											// 
		bAlarm5			:= FALSE, 											//
		bAlarm6			:= FALSE,                                           //
		bAlarm7			:= FALSE,                                           //
		bAlarm8			:= FALSE,                                           //
		bAlarm9			:= FALSE,                                           //
		bAlarm10		:= FALSE,                                           //
		bAlarm11		:= FALSE,                                           //
		bAlarm12		:= FALSE,                                           //
		bAlarm13		:= FALSE,                                           //
		bAlarm14		:= FALSE,                                           //
		bAlarm15		:= FALSE,                                           //
		wAlarmCode		=>MesDataExd.MesData.MesWarningCode);

// EVENT CODE //
	FB_AlarmCodeManager(
		bAlarm1			:=FALSE, 											// 
		bAlarm2			:=FALSE, 											// 
		bAlarm3			:=FALSE, 											// 
		bAlarm4			:=FALSE, 											// 
		bAlarm5			:=FALSE, 											//
		bAlarm6			:=FALSE, 											//
		bAlarm7			:=FALSE, 											//
		bAlarm8			:=FALSE, 											//
		bAlarm9			:=FALSE, 											//
		bAlarm10		:=FALSE, 											//
		bAlarm11		:=FALSE, 											//
		bAlarm12		:=FALSE, 											//
		bAlarm13		:=FALSE, 											//
		bAlarm14		:=FALSE, 											//
		bAlarm15		:=FALSE, 											//
		wAlarmCode		=>MesDataExd.MesData.MesEventCode);
END_METHOD

END_FUNCTION_BLOCK

// ---- 04_Application/MAIN/POU.TcPOU
FUNCTION_BLOCK POU
VAR_INPUT
END_VAR
VAR_OUTPUT
END_VAR
VAR
END_VAR

END_FUNCTION_BLOCK
